//{attribute 'qualified_only'}
{attribute 'strict'}
{attribute 'to_string'}
TYPE MachineState :
(
	off   := 0, 
	on    := 1
	//error := 2
);
END_TYPE

(* stored: Version 1.1.0.1
   DUT MachineState: Id {efb98ac1-2c38-42d6-8584-62264cb5e132} *)
